FUNCTION_BLOCK FB_XmlPersistentEventStorage IMPLEMENTS I_PersistentEventStorage
VAR_INPUT
END_VAR
VAR_OUTPUT
END_VAR
VAR
END_VAR

//

METHOD StoreEvent
VAR_INPUT
	stEvent	: ST_Event;
END_VAR
END_METHOD

END_FUNCTION_BLOCK

(* stored: Version 1.1.0.1, ProductVersion 3.1.4024.12
   POU FB_XmlPersistentEventStorage: Id {e3123194-14a3-47a7-8c04-689e285d04b2}, SpecialFunc None
   Method StoreEvent: Id {68fa816d-474b-490e-afc3-2cfd852098d7} *)
